FUNCTION_BLOCK NodeFinder (* Composite Function Block Type *)
  (* Standard: 61499-2 *)
  (* Version 0.0, 2/5/2024, midxav, template *)
  PACKAGE Main;
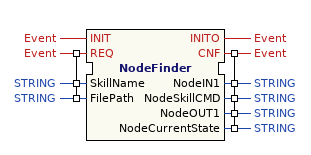
  EVENT_INPUT
    INIT;
    REQ WITH SkillName, FilePath;
  END_EVENT
  EVENT_OUTPUT
    INITO;
    CNF WITH NodeIN1, NodeSkillCMD, NodeOUT1, NodeCurrentState;
  END_EVENT
  VAR_INPUT
    SkillName : STRING;
    FilePath : STRING;
  END_VAR
  VAR_OUTPUT
    NodeIN1 : STRING;
    NodeSkillCMD : STRING;
    NodeOUT1 : STRING;
    NodeCurrentState : STRING;
  END_VAR
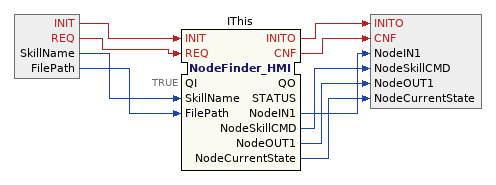
  FBS
    IThis : NodeFinder_HMI(QI := TRUE);
  END_FBS
  EVENT_CONNECTIONS
    IThis.INITO TO INITO;
    IThis.CNF TO CNF;
    INIT TO IThis.INIT;
    REQ TO IThis.REQ;
  END_CONNECTIONS
  DATA_CONNECTIONS
    SkillName TO IThis.SkillName;
    FilePath TO IThis.FilePath;
    IThis.NodeIN1 TO NodeIN1;
    IThis.NodeSkillCMD TO NodeSkillCMD;
    IThis.NodeOUT1 TO NodeOUT1;
    IThis.NodeCurrentState TO NodeCurrentState;
  END_CONNECTIONS
END_FUNCTION_BLOCK
